TYPE ST_ShuttleRecipe :
STRUCT
		Velocity     : LREAL;
        Acceleration : LREAL;
		CassettePosition : LREAL;
		ToolPosition : LREAL;
END_STRUCT
END_TYPE

(* stored: Version 1.1.0.1, ProductVersion 3.1.4024.12
   DUT ST_ShuttleRecipe: Id {bd4f506a-05d2-4636-bdea-d2942d9245e7} *)
